FUNCTION_BLOCK Mixing EXTENDS BaseState
VAR_INPUT
END_VAR
VAR_OUTPUT
END_VAR
VAR
	InternalMixingTime : TIME;
END_VAR

METHOD mIrun : BOOL
StateTimer(IN:=TRUE, PT:=InternalMixingTime);
BasePointer^.MachineFlagsAccessI.pMixing := TRUE;
IF StateTimer.Q THEN
	mNextState();
	BasePointer^.MachineFlagsAccessI.pMixing := FALSE;
	StateTimer(IN:=FALSE);
END_IF
END_METHOD

METHOD mStateInit : BOOL
VAR_INPUT
	MixingTime : TIME;
END_VAR
InternalMixingTime := MixingTime;
END_METHOD

END_FUNCTION_BLOCK

(* stored: Version 1.1.0.1, ProductVersion 3.1.4024.12
   POU Mixing: Id {7c986a47-0b45-4a7c-91ca-7ac3ed8c508a}, SpecialFunc None
   Method mIrun: Id {399c1e34-8270-4677-a09c-a2fe7c8983ec}
   Method mStateInit: Id {a9c3c502-1ea6-48c7-a6be-b40ac9c75059} *)
